// TIA Portal V17 export
// export: Created 2024-09-02T12:50:21.0608261Z, ExportSetting WithDefaults, DisplayName Totally Integrated Automation Portal, DisplayVersion V17, DisplayName TIA Portal Openness, DisplayVersion V17, DisplayName TIA Portal Version Control Interface, DisplayVersion V17, DisplayName STEP 7 Professional, DisplayVersion V17, DisplayName STEP 7 Safety, DisplayVersion V17, DisplayName WinCC Professional, DisplayVersion V17
FUNCTION "AnwFC0_FG02_Management_SLG2_OP70" : Void   // FC1014, LAD
TITLE = Administration Moby / Verwaltung Moby
{ S7_Optimized_Access := 'TRUE' }
AUTHOR : OlegFuehrus
FAMILY : MOBY
NAME : OlegFuehrus
VERSION : 0.1
// stored: AutoNumber false, IsIECCheckEnabled false, SetENOAutomatically false, UDAEnableTagReadback false
   VAR_TEMP
      Motion_Release : Bool;   // Bewegungsfreigabe / Motion permit
      Hand : Bool;   // Handbetrieb / Manual mode
      Auto : Bool;   // Automatikbetrieb / Automatic mode
      _VKE0 : Bool;   // VKE 0
      _VKE1 : Bool;   // VKE 1
      _ASM_ID : Int;   // Hardware ID ASM
      _ASM_ADR : Int;   // Hardwareadresse ASM / Hardware address ASM
      _ASM_CHANNEL : Int;   // Kanalnummer ASM / Channel number ASM
      _Evaluation_finished : Bool;   // Auswertung Fertig / Evaluation finished
      _Backbilling_finished : Bool;   // Rückberechnung Fertig / Recalculation Finished
   END_VAR
BEGIN

REGION Network 1: Parameters: SLG no. / Parameter: SLG-Nr.
   // will change / wird sich ändern
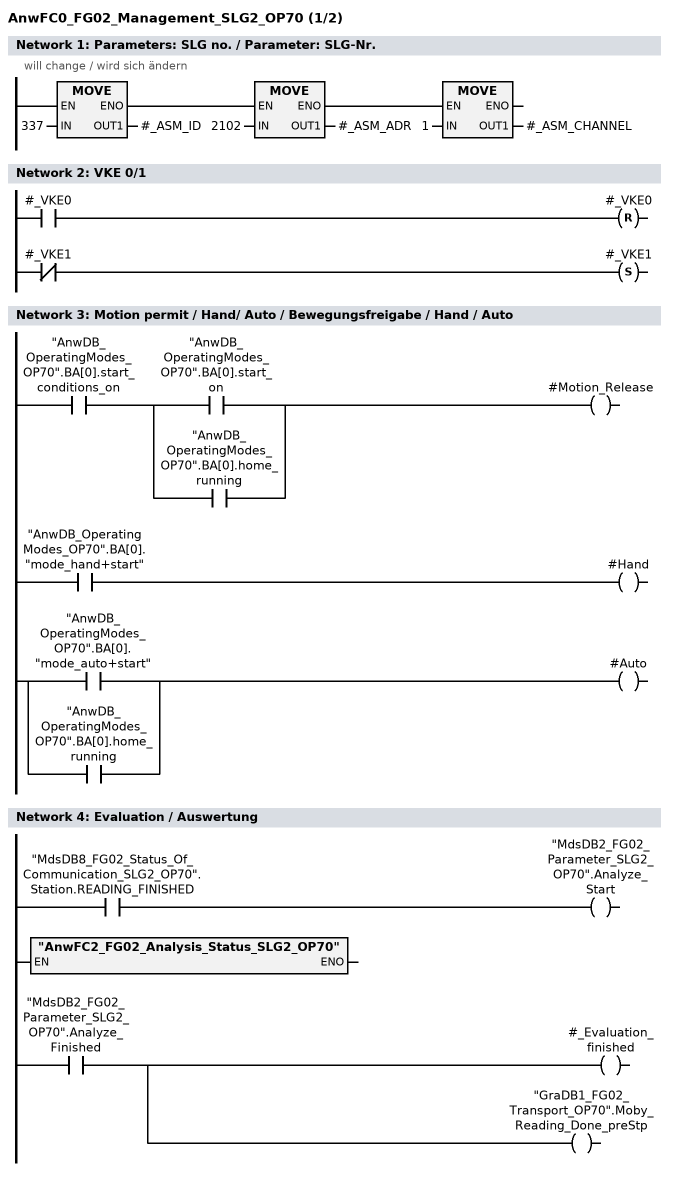
   RUNG wire#powerrail
      { S7_GenerateENO := "TRUE" } Move(in := 337, out1 => #_ASM_ID)
      { S7_GenerateENO := "TRUE" } Move(in := 2102, out1 => #_ASM_ADR)
      { S7_GenerateENO := "TRUE" } Move(in := 1, out1 => #_ASM_CHANNEL)
   END_RUNG
   // the same network as SCL:
   // ENO of a box is taken as its EN; it also drops when the box reports an error
   #_ASM_ID := 337;
   #_ASM_ADR := 2102;
   #_ASM_CHANNEL := 1;
END_REGION

REGION Network 2: VKE 0/1
   RUNG wire#powerrail
      Contact( #_VKE0 )
      R_Coil( #_VKE0 )
   END_RUNG
   RUNG wire#powerrail
      I_Contact( #_VKE1 )
      S_Coil( #_VKE1 )
   END_RUNG
   // the same network as SCL:
   IF #_VKE0 THEN #_VKE0 := FALSE; END_IF;
   IF NOT #_VKE1 THEN #_VKE1 := TRUE; END_IF;
END_REGION

REGION Network 3: Motion permit / Hand/ Auto / Bewegungsfreigabe / Hand / Auto
   RUNG wire#powerrail
      Contact( "AnwDB_OperatingModes_OP70".BA[0].start_conditions_on )
      wire#w1
      Contact( "AnwDB_OperatingModes_OP70".BA[0].start_on )
      wire#w2
      Coil( #Motion_Release )
   END_RUNG
   RUNG wire#w1
      Contact( "AnwDB_OperatingModes_OP70".BA[0].home_running )
   END_RUNG wire#w2
   RUNG wire#powerrail
      Contact( "AnwDB_OperatingModes_OP70".BA[0]."mode_hand+start" )
      Coil( #Hand )
   END_RUNG
   RUNG wire#powerrail
      Contact( "AnwDB_OperatingModes_OP70".BA[0]."mode_auto+start" )
      wire#w3
      Coil( #Auto )
   END_RUNG
   RUNG wire#powerrail
      Contact( "AnwDB_OperatingModes_OP70".BA[0].home_running )
   END_RUNG wire#w3
   // the same network as SCL:
   #Motion_Release := "AnwDB_OperatingModes_OP70".BA[0].start_conditions_on AND ("AnwDB_OperatingModes_OP70".BA[0].start_on OR "AnwDB_OperatingModes_OP70".BA[0].home_running);
   #Hand := "AnwDB_OperatingModes_OP70".BA[0]."mode_hand+start";
   #Auto := "AnwDB_OperatingModes_OP70".BA[0]."mode_auto+start" OR "AnwDB_OperatingModes_OP70".BA[0].home_running;
END_REGION

REGION Network 4: Evaluation / Auswertung
   RUNG wire#powerrail
      Contact( "MdsDB8_FG02_Status_Of_Communication_SLG2_OP70".Station.READING_FINISHED )
      Coil( "MdsDB2_FG02_Parameter_SLG2_OP70".Analyze_Start )
   END_RUNG
   RUNG wire#powerrail
      "AnwFC2_FG02_Analysis_Status_SLG2_OP70"()
   END_RUNG
   RUNG wire#powerrail
      Contact( "MdsDB2_FG02_Parameter_SLG2_OP70".Analyze_Finished )
      wire#w1
      Coil( #_Evaluation_finished )
   END_RUNG
   RUNG wire#w1
      Coil( "GraDB1_FG02_Transport_OP70".Moby_Reading_Done_preStp )
   END_RUNG
   // the same network as SCL:
   "MdsDB2_FG02_Parameter_SLG2_OP70".Analyze_Start := "MdsDB8_FG02_Status_Of_Communication_SLG2_OP70".Station.READING_FINISHED;
   "AnwFC2_FG02_Analysis_Status_SLG2_OP70"();
   #_Evaluation_finished := "MdsDB2_FG02_Parameter_SLG2_OP70".Analyze_Finished;
   "GraDB1_FG02_Transport_OP70".Moby_Reading_Done_preStp := "MdsDB2_FG02_Parameter_SLG2_OP70".Analyze_Finished;
END_REGION

REGION Network 5: Recalculation / Rückberechnung
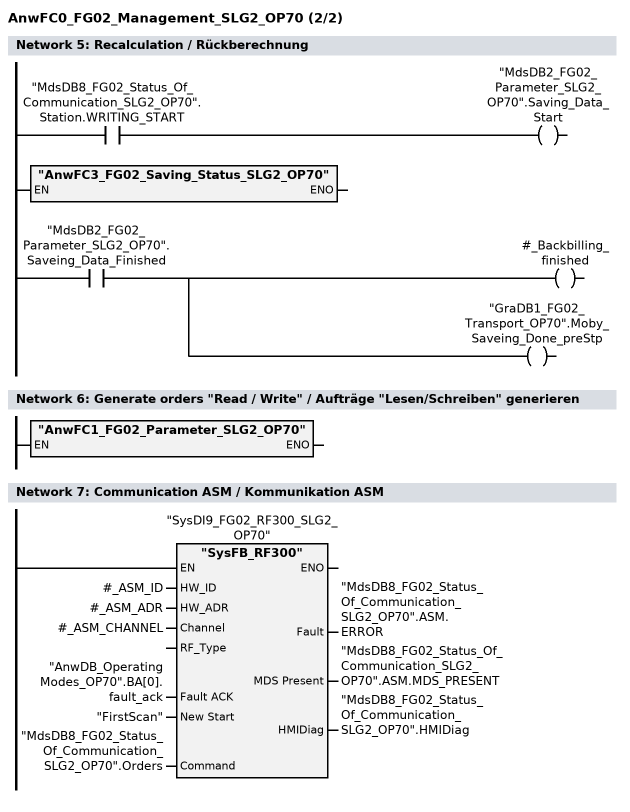
   RUNG wire#powerrail
      Contact( "MdsDB8_FG02_Status_Of_Communication_SLG2_OP70".Station.WRITING_START )
      Coil( "MdsDB2_FG02_Parameter_SLG2_OP70".Saving_Data_Start )
   END_RUNG
   RUNG wire#powerrail
      "AnwFC3_FG02_Saving_Status_SLG2_OP70"()
   END_RUNG
   RUNG wire#powerrail
      Contact( "MdsDB2_FG02_Parameter_SLG2_OP70".Saveing_Data_Finished )
      wire#w1
      Coil( #_Backbilling_finished )
   END_RUNG
   RUNG wire#w1
      Coil( "GraDB1_FG02_Transport_OP70".Moby_Saveing_Done_preStp )
   END_RUNG
   // the same network as SCL:
   "MdsDB2_FG02_Parameter_SLG2_OP70".Saving_Data_Start := "MdsDB8_FG02_Status_Of_Communication_SLG2_OP70".Station.WRITING_START;
   "AnwFC3_FG02_Saving_Status_SLG2_OP70"();
   #_Backbilling_finished := "MdsDB2_FG02_Parameter_SLG2_OP70".Saveing_Data_Finished;
   "GraDB1_FG02_Transport_OP70".Moby_Saveing_Done_preStp := "MdsDB2_FG02_Parameter_SLG2_OP70".Saveing_Data_Finished;
END_REGION

REGION Network 6: Generate orders "Read / Write" / Aufträge "Lesen/Schreiben" generieren
   RUNG wire#powerrail
      "AnwFC1_FG02_Parameter_SLG2_OP70"()
   END_RUNG
   // the same network as SCL:
   "AnwFC1_FG02_Parameter_SLG2_OP70"();
END_REGION

REGION Network 7: Communication ASM / Kommunikation ASM
   RUNG wire#powerrail
      "SysDI9_FG02_RF300_SLG2_OP70"(HW_ID := #_ASM_ID, HW_ADR := #_ASM_ADR, Channel := #_ASM_CHANNEL, RF_Type :=, "Fault ACK" := "AnwDB_OperatingModes_OP70".BA[0].fault_ack, "New Start" := "FirstScan", Command := "MdsDB8_FG02_Status_Of_Communication_SLG2_OP70".Orders, Fault => "MdsDB8_FG02_Status_Of_Communication_SLG2_OP70".ASM.ERROR, "MDS Present" => "MdsDB8_FG02_Status_Of_Communication_SLG2_OP70".ASM.MDS_PRESENT, HMIDiag => "MdsDB8_FG02_Status_Of_Communication_SLG2_OP70".HMIDiag)
   END_RUNG
   // the same network as SCL:
   "SysDI9_FG02_RF300_SLG2_OP70"(HW_ID := #_ASM_ID,   // "SysFB_RF300"
                           HW_ADR := #_ASM_ADR,
                           Channel := #_ASM_CHANNEL,
                           "Fault ACK" := "AnwDB_OperatingModes_OP70".BA[0].fault_ack,
                           "New Start" := "FirstScan",
                           Command := "MdsDB8_FG02_Status_Of_Communication_SLG2_OP70".Orders,
                           Fault => "MdsDB8_FG02_Status_Of_Communication_SLG2_OP70".ASM.ERROR,
                           "MDS Present" => "MdsDB8_FG02_Status_Of_Communication_SLG2_OP70".ASM.MDS_PRESENT,
                           HMIDiag => "MdsDB8_FG02_Status_Of_Communication_SLG2_OP70".HMIDiag);
END_REGION
END_FUNCTION
